ABB RobotStudio station: Practica2_ej2_extra1.rspag

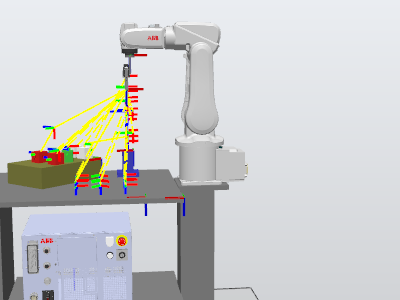
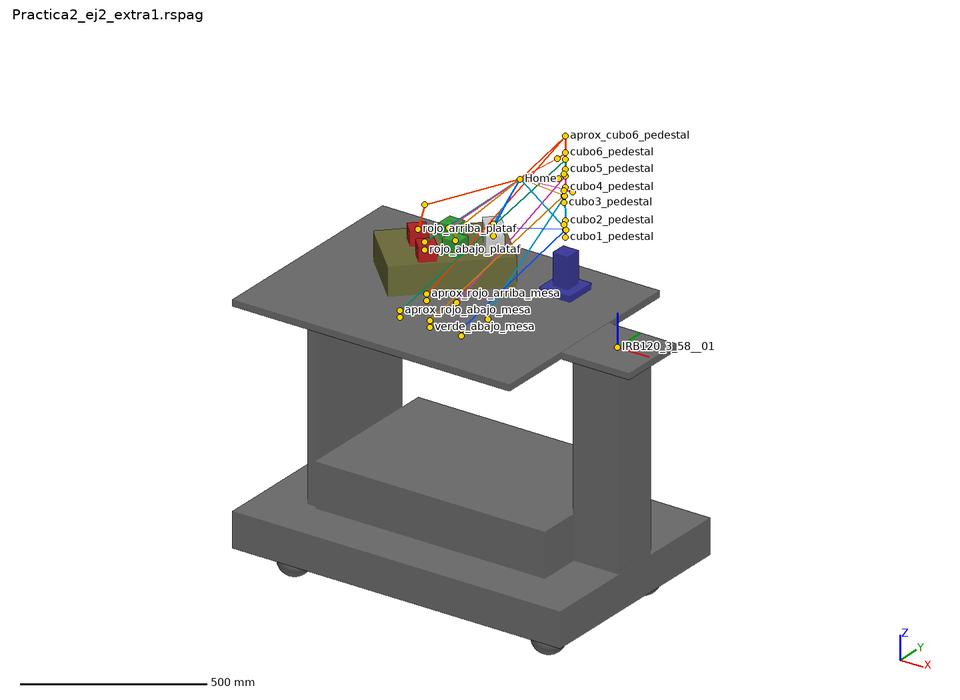
[picture v1: parts stored in the station drawn from their meshes, with robot base, taught points and paths (robot models come from the ABB library and are not in the file)]
--- station ---
Station Practica2_1920 (saved by RobotStudio 24.4.11080.0)
Controller Controlador_IRC5, task T_ROB1: task frame (RAPID world) sits at (560, 0, 840) mm, rotated rx 0 ry 0 rz 180 deg in the station
Controller Controlador_IRC5
  mechanical unit ROB_1: IRB120_3_58__01, 6 joints, base frame (0, 0, 0) mm
Layout (positions relative to the parent item):
  - Pinza_schunk_SGB50 [mechanism, from Libraries\Pinza_schunk_SGB50.rslib] at (258, 0, 1398) mm, rotated rx 180 ry 0 rz 0 deg; joint values [0, 0.1745, -0.1745] (rad or m)
  - Mesa del robot [part], size 1127.5 x 700 x 840 mm
  - Cubo XYZ 50 mm 2 [part] at (-54.74, 116.46, 930) mm, rotated rx 0 ry 0 rz 90 deg, size 50 x 50 x 50 mm
  - Cubo XYZ 50 mm 3 [part] at (7.57, 171.09, 931.86) mm, rotated rx 0 ry 0 rz 45 deg, size 50 x 50 x 50 mm
  - Cubo XYZ 50 mm 4 [part] at (-100.89, 1.6, 929.03) mm, rotated rx 0 ry 0 rz -45 deg, size 50 x 50 x 50 mm
  - Cubo XYZ 50 mm 5 [part] at (5.14, 45.89, 928.53) mm, rotated rx 0 ry 0 rz 90 deg, size 50 x 50 x 50 mm
  - Cubo XYZ 50 mm 6 [part] at (54.86, 109.05, 933.24) mm, rotated rx 0 ry 0 rz 45 deg, size 50 x 50 x 50 mm
  - Cubo XYZ 50 mm 1 [part] at (-175.7, 68.89, 928.24) mm, rotated rx 0 ry 0 rz -45 deg, size 50 x 50 x 50 mm
  - Soporte para elevar los cubos  [part] at (200, 150, 840) mm, size 100 x 100 x 120 mm
  - IRC5_Compact [part, from %ABB.RobotStudio.Models.IRC5%\IRC5_Compact__02.rslib] at (-200, -200, 350) mm
  - Soporte para el controlador [part], size 750 x 480 x 150 mm
  - IRB120_3_58__01 [mechanism, from %ABB.RobotStudio.Models.IRB120%\IRB120_3_58_G_01.rslib] at (560, 0, 840) mm, rotated rx 0 ry 0 rz 180 deg; joint values [0, 0, 0, 0, 1.5708, 0] (rad or m)
  - caja [part], size 406.6 x 406.6 x 90 mm
Attachment: Soporte para el controlador is attached to Mesa del robot
Attachment: Pinza_schunk_SGB50 is attached to IRB120_3_58__01 / Link6
EventTableEntry 2988: Group=, Trigger=D16_O 2989, Actions=[EventTableActionMechanicalPose 2990, EventTableActionAttach 2991], Comment=, ActivationMode=2, Cyclic=false
EventTableTriggerIO 2989: IOValue=[1], IRC5Controller=? -1, Operator=0, SignalSource=Controlador_IRC5 2505
EventTableActionMechanicalPose 2990: VirtualSignal=, Mechanism=Pinza_schunk_SGB50 1474, ToPoseName=HomePosition, VirtualSignalValue=[1]
EventTableActionAttach 2991: AttachmentParent=Pinza_schunk_SGB50 1474, AttachmentChild=? -1, MountObject=false, Offset=[X=1, Y=0, Z=0, W=0, X=0, Y=1, Z=0, W=0, X=0, Y=0, Z=1, W=0, X=0, Y=0, Z=0, W=1], FlangeIndext=0, FindNearest=true
EventTableEntry 2992: Group=, Trigger=D16_O 2993, Actions=[EventTableActionMechanicalPose 2994, EventTableActionDetach 2995], Comment=, ActivationMode=2, Cyclic=false
EventTableTriggerIO 2993: IOValue=[0], IRC5Controller=? -1, Operator=0, SignalSource=Controlador_IRC5 2505
EventTableActionMechanicalPose 2994: VirtualSignal=, Mechanism=Pinza_schunk_SGB50 1474, ToPoseName=Abierto, VirtualSignalValue=[1]
EventTableActionDetach 2995: AttachmentParent=Pinza_schunk_SGB50 1474, AttachmentChild=? -1
EventTableTriggerIO 3053: IOValue=[1], IRC5Controller=? -1, Operator=0, SignalSource=Controlador_IRC5 2505
EventTableTriggerIO 3054: IOValue=[1], IRC5Controller=? -1, Operator=0, SignalSource=Controlador_IRC5 2505
EventTableTriggerIO 3055: IOValue=[1], IRC5Controller=? -1, Operator=0, SignalSource=Controlador_IRC5 2505
EventTableTriggerIO 3056: IOValue=[1], IRC5Controller=? -1, Operator=0, SignalSource=Controlador_IRC5 2505
EventTableTriggerIO 3057: IOValue=[1], IRC5Controller=? -1, Operator=0, SignalSource=Controlador_IRC5 2505
EventTableTriggerIO 3058: IOValue=[1], IRC5Controller=? -1, Operator=0, SignalSource=Controlador_IRC5 2505
EventTableTriggerIO 3059: IOValue=[1], IRC5Controller=? -1, Operator=0, SignalSource=Controlador_IRC5 2505
EventTableTriggerIO 3060: IOValue=[1], IRC5Controller=? -1, Operator=0, SignalSource=Controlador_IRC5 2505
EventTableTriggerIO 3061: IOValue=[1], IRC5Controller=? -1, Operator=0, SignalSource=Controlador_IRC5 2505
EventTableTriggerIO 3062: IOValue=[1], IRC5Controller=? -1, Operator=0, SignalSource=Controlador_IRC5 2505
EventTableTriggerIO 3063: IOValue=[1], IRC5Controller=? -1, Operator=0, SignalSource=Controlador_IRC5 2505
EventTableTriggerIO 3064: IOValue=[1], IRC5Controller=? -1, Operator=0, SignalSource=Controlador_IRC5 2505
EventTableTriggerIO 3065: IOValue=[0], IRC5Controller=? -1, Operator=0, SignalSource=Controlador_IRC5 2505
EventTableTriggerIO 3066: IOValue=[0], IRC5Controller=? -1, Operator=0, SignalSource=Controlador_IRC5 2505
EventTableTriggerIO 3067: IOValue=[0], IRC5Controller=? -1, Operator=0, SignalSource=Controlador_IRC5 2505
EventTableTriggerIO 3068: IOValue=[0], IRC5Controller=? -1, Operator=0, SignalSource=Controlador_IRC5 2505
EventTableTriggerIO 3069: IOValue=[0], IRC5Controller=? -1, Operator=0, SignalSource=Controlador_IRC5 2505
EventTableTriggerIO 3070: IOValue=[0], IRC5Controller=? -1, Operator=0, SignalSource=Controlador_IRC5 2505
EventTableTriggerIO 3071: IOValue=[0], IRC5Controller=? -1, Operator=0, SignalSource=Controlador_IRC5 2505
EventTableTriggerIO 3072: IOValue=[0], IRC5Controller=? -1, Operator=0, SignalSource=Controlador_IRC5 2505
EventTableTriggerIO 3073: IOValue=[0], IRC5Controller=? -1, Operator=0, SignalSource=Controlador_IRC5 2505
EventTableTriggerIO 3074: IOValue=[0], IRC5Controller=? -1, Operator=0, SignalSource=Controlador_IRC5 2505
EventTableTriggerIO 3075: IOValue=[0], IRC5Controller=? -1, Operator=0, SignalSource=Controlador_IRC5 2505
EventTableTriggerIO 3076: IOValue=[0], IRC5Controller=? -1, Operator=0, SignalSource=Controlador_IRC5 2505
EventTableTriggerIO 3176: IOValue=[1], IRC5Controller=? -1, Operator=0, SignalSource=Controlador_IRC5 2505
EventTableTriggerIO 3177: IOValue=[1], IRC5Controller=? -1, Operator=0, SignalSource=Controlador_IRC5 2505
EventTableTriggerIO 3178: IOValue=[1], IRC5Controller=? -1, Operator=0, SignalSource=Controlador_IRC5 2505
EventTableTriggerIO 3179: IOValue=[1], IRC5Controller=? -1, Operator=0, SignalSource=Controlador_IRC5 2505
EventTableTriggerIO 3180: IOValue=[1], IRC5Controller=? -1, Operator=0, SignalSource=Controlador_IRC5 2505
EventTableTriggerIO 3181: IOValue=[0], IRC5Controller=? -1, Operator=0, SignalSource=Controlador_IRC5 2505
EventTableTriggerIO 3182: IOValue=[0], IRC5Controller=? -1, Operator=0, SignalSource=Controlador_IRC5 2505
EventTableTriggerIO 3183: IOValue=[0], IRC5Controller=? -1, Operator=0, SignalSource=Controlador_IRC5 2505
EventTableTriggerIO 3184: IOValue=[0], IRC5Controller=? -1, Operator=0, SignalSource=Controlador_IRC5 2505
EventTableTriggerIO 3185: IOValue=[0], IRC5Controller=? -1, Operator=0, SignalSource=Controlador_IRC5 2505
EventTableTriggerIO 3333: IOValue=[1], IRC5Controller=? -1, Operator=0, SignalSource=Controlador_IRC5 2505
EventTableTriggerIO 3334: IOValue=[1], IRC5Controller=? -1, Operator=0, SignalSource=Controlador_IRC5 2505
EventTableTriggerIO 3335: IOValue=[1], IRC5Controller=? -1, Operator=0, SignalSource=Controlador_IRC5 2505
EventTableTriggerIO 3336: IOValue=[1], IRC5Controller=? -1, Operator=0, SignalSource=Controlador_IRC5 2505
EventTableTriggerIO 3337: IOValue=[1], IRC5Controller=? -1, Operator=0, SignalSource=Controlador_IRC5 2505
EventTableTriggerIO 3338: IOValue=[1], IRC5Controller=? -1, Operator=0, SignalSource=Controlador_IRC5 2505
EventTableTriggerIO 3339: IOValue=[0], IRC5Controller=? -1, Operator=0, SignalSource=Controlador_IRC5 2505
EventTableTriggerIO 3340: IOValue=[0], IRC5Controller=? -1, Operator=0, SignalSource=Controlador_IRC5 2505
EventTableTriggerIO 3341: IOValue=[0], IRC5Controller=? -1, Operator=0, SignalSource=Controlador_IRC5 2505
EventTableTriggerIO 3342: IOValue=[0], IRC5Controller=? -1, Operator=0, SignalSource=Controlador_IRC5 2505
EventTableTriggerIO 3343: IOValue=[0], IRC5Controller=? -1, Operator=0, SignalSource=Controlador_IRC5 2505
EventTableTriggerIO 3344: IOValue=[0], IRC5Controller=? -1, Operator=0, SignalSource=Controlador_IRC5 2505
EventTableTriggerIO 3580: IOValue=[1], IRC5Controller=? -1, Operator=0, SignalSource=Controlador_IRC5 2505
EventTableTriggerIO 3581: IOValue=[1], IRC5Controller=? -1, Operator=0, SignalSource=Controlador_IRC5 2505
EventTableTriggerIO 3582: IOValue=[1], IRC5Controller=? -1, Operator=0, SignalSource=Controlador_IRC5 2505
EventTableTriggerIO 3583: IOValue=[1], IRC5Controller=? -1, Operator=0, SignalSource=Controlador_IRC5 2505
EventTableTriggerIO 3584: IOValue=[1], IRC5Controller=? -1, Operator=0, SignalSource=Controlador_IRC5 2505
EventTableTriggerIO 3585: IOValue=[1], IRC5Controller=? -1, Operator=0, SignalSource=Controlador_IRC5 2505
EventTableTriggerIO 3586: IOValue=[1], IRC5Controller=? -1, Operator=0, SignalSource=Controlador_IRC5 2505
EventTableTriggerIO 3587: IOValue=[1], IRC5Controller=? -1, Operator=0, SignalSource=Controlador_IRC5 2505
EventTableTriggerIO 3588: IOValue=[1], IRC5Controller=? -1, Operator=0, SignalSource=Controlador_IRC5 2505
EventTableTriggerIO 3589: IOValue=[1], IRC5Controller=? -1, Operator=0, SignalSource=Controlador_IRC5 2505
EventTableTriggerIO 3590: IOValue=[0], IRC5Controller=? -1, Operator=0, SignalSource=Controlador_IRC5 2505
EventTableTriggerIO 3591: IOValue=[0], IRC5Controller=? -1, Operator=0, SignalSource=Controlador_IRC5 2505
EventTableTriggerIO 3592: IOValue=[0], IRC5Controller=? -1, Operator=0, SignalSource=Controlador_IRC5 2505
EventTableTriggerIO 3593: IOValue=[0], IRC5Controller=? -1, Operator=0, SignalSource=Controlador_IRC5 2505
EventTableTriggerIO 3594: IOValue=[0], IRC5Controller=? -1, Operator=0, SignalSource=Controlador_IRC5 2505
EventTableTriggerIO 3595: IOValue=[0], IRC5Controller=? -1, Operator=0, SignalSource=Controlador_IRC5 2505
EventTableTriggerIO 3596: IOValue=[0], IRC5Controller=? -1, Operator=0, SignalSource=Controlador_IRC5 2505
EventTableTriggerIO 3597: IOValue=[0], IRC5Controller=? -1, Operator=0, SignalSource=Controlador_IRC5 2505
EventTableTriggerIO 3598: IOValue=[0], IRC5Controller=? -1, Operator=0, SignalSource=Controlador_IRC5 2505
EventTableTriggerIO 3599: IOValue=[0], IRC5Controller=? -1, Operator=0, SignalSource=Controlador_IRC5 2505
EventTableTriggerIO 3839: IOValue=[1], IRC5Controller=? -1, Operator=0, SignalSource=Controlador_IRC5 2505
EventTableTriggerIO 3840: IOValue=[1], IRC5Controller=? -1, Operator=0, SignalSource=Controlador_IRC5 2505
EventTableTriggerIO 3841: IOValue=[1], IRC5Controller=? -1, Operator=0, SignalSource=Controlador_IRC5 2505
EventTableTriggerIO 3842: IOValue=[1], IRC5Controller=? -1, Operator=0, SignalSource=Controlador_IRC5 2505
EventTableTriggerIO 3843: IOValue=[1], IRC5Controller=? -1, Operator=0, SignalSource=Controlador_IRC5 2505
EventTableTriggerIO 3844: IOValue=[1], IRC5Controller=? -1, Operator=0, SignalSource=Controlador_IRC5 2505
EventTableTriggerIO 3845: IOValue=[1], IRC5Controller=? -1, Operator=0, SignalSource=Controlador_IRC5 2505
EventTableTriggerIO 3846: IOValue=[1], IRC5Controller=? -1, Operator=0, SignalSource=Controlador_IRC5 2505
EventTableTriggerIO 3847: IOValue=[1], IRC5Controller=? -1, Operator=0, SignalSource=Controlador_IRC5 2505
EventTableTriggerIO 3848: IOValue=[1], IRC5Controller=? -1, Operator=0, SignalSource=Controlador_IRC5 2505
EventTableTriggerIO 3849: IOValue=[1], IRC5Controller=? -1, Operator=0, SignalSource=Controlador_IRC5 2505
EventTableTriggerIO 3850: IOValue=[1], IRC5Controller=? -1, Operator=0, SignalSource=Controlador_IRC5 2505
EventTableTriggerIO 3851: IOValue=[1], IRC5Controller=? -1, Operator=0, SignalSource=Controlador_IRC5 2505
EventTableTriggerIO 3852: IOValue=[1], IRC5Controller=? -1, Operator=0, SignalSource=Controlador_IRC5 2505
EventTableTriggerIO 3853: IOValue=[1], IRC5Controller=? -1, Operator=0, SignalSource=Controlador_IRC5 2505
EventTableTriggerIO 3854: IOValue=[0], IRC5Controller=? -1, Operator=0, SignalSource=Controlador_IRC5 2505
EventTableTriggerIO 3855: IOValue=[0], IRC5Controller=? -1, Operator=0, SignalSource=Controlador_IRC5 2505
EventTableTriggerIO 3856: IOValue=[0], IRC5Controller=? -1, Operator=0, SignalSource=Controlador_IRC5 2505
EventTableTriggerIO 3857: IOValue=[0], IRC5Controller=? -1, Operator=0, SignalSource=Controlador_IRC5 2505
EventTableTriggerIO 3858: IOValue=[0], IRC5Controller=? -1, Operator=0, SignalSource=Controlador_IRC5 2505
EventTableTriggerIO 3859: IOValue=[0], IRC5Controller=? -1, Operator=0, SignalSource=Controlador_IRC5 2505
EventTableTriggerIO 3860: IOValue=[0], IRC5Controller=? -1, Operator=0, SignalSource=Controlador_IRC5 2505
EventTableTriggerIO 3861: IOValue=[0], IRC5Controller=? -1, Operator=0, SignalSource=Controlador_IRC5 2505
EventTableTriggerIO 3862: IOValue=[0], IRC5Controller=? -1, Operator=0, SignalSource=Controlador_IRC5 2505
EventTableTriggerIO 3863: IOValue=[0], IRC5Controller=? -1, Operator=0, SignalSource=Controlador_IRC5 2505
EventTableTriggerIO 3864: IOValue=[0], IRC5Controller=? -1, Operator=0, SignalSource=Controlador_IRC5 2505
EventTableTriggerIO 3865: IOValue=[0], IRC5Controller=? -1, Operator=0, SignalSource=Controlador_IRC5 2505
EventTableTriggerIO 3866: IOValue=[0], IRC5Controller=? -1, Operator=0, SignalSource=Controlador_IRC5 2505
EventTableTriggerIO 3867: IOValue=[0], IRC5Controller=? -1, Operator=0, SignalSource=Controlador_IRC5 2505
EventTableTriggerIO 3868: IOValue=[0], IRC5Controller=? -1, Operator=0, SignalSource=Controlador_IRC5 2505
EventTableTriggerIO 4020: IOValue=[1], IRC5Controller=? -1, Operator=0, SignalSource=Controlador_IRC5 2505
EventTableTriggerIO 4021: IOValue=[1], IRC5Controller=? -1, Operator=0, SignalSource=Controlador_IRC5 2505
EventTableTriggerIO 4022: IOValue=[1], IRC5Controller=? -1, Operator=0, SignalSource=Controlador_IRC5 2505
EventTableTriggerIO 4023: IOValue=[1], IRC5Controller=? -1, Operator=0, SignalSource=Controlador_IRC5 2505
EventTableTriggerIO 4024: IOValue=[1], IRC5Controller=? -1, Operator=0, SignalSource=Controlador_IRC5 2505
EventTableTriggerIO 4025: IOValue=[1], IRC5Controller=? -1, Operator=0, SignalSource=Controlador_IRC5 2505
EventTableTriggerIO 4026: IOValue=[0], IRC5Controller=? -1, Operator=0, SignalSource=Controlador_IRC5 2505
EventTableTriggerIO 4027: IOValue=[0], IRC5Controller=? -1, Operator=0, SignalSource=Controlador_IRC5 2505
EventTableTriggerIO 4028: IOValue=[0], IRC5Controller=? -1, Operator=0, SignalSource=Controlador_IRC5 2505
EventTableTriggerIO 4029: IOValue=[0], IRC5Controller=? -1, Operator=0, SignalSource=Controlador_IRC5 2505
EventTableTriggerIO 4030: IOValue=[0], IRC5Controller=? -1, Operator=0, SignalSource=Controlador_IRC5 2505
EventTableTriggerIO 4031: IOValue=[0], IRC5Controller=? -1, Operator=0, SignalSource=Controlador_IRC5 2505
EventTableTriggerIO 4133: IOValue=[1], IRC5Controller=? -1, Operator=0, SignalSource=Controlador_IRC5 2505
EventTableTriggerIO 4134: IOValue=[1], IRC5Controller=? -1, Operator=0, SignalSource=Controlador_IRC5 2505
EventTableTriggerIO 4135: IOValue=[0], IRC5Controller=? -1, Operator=0, SignalSource=Controlador_IRC5 2505
EventTableTriggerIO 4136: IOValue=[0], IRC5Controller=? -1, Operator=0, SignalSource=Controlador_IRC5 2505
EventTableTriggerIO 4229: IOValue=[1], IRC5Controller=? -1, Operator=0, SignalSource=Controlador_IRC5 2505
EventTableTriggerIO 4230: IOValue=[1], IRC5Controller=? -1, Operator=0, SignalSource=Controlador_IRC5 2505
EventTableTriggerIO 4231: IOValue=[1], IRC5Controller=? -1, Operator=0, SignalSource=Controlador_IRC5 2505
EventTableTriggerIO 4232: IOValue=[1], IRC5Controller=? -1, Operator=0, SignalSource=Controlador_IRC5 2505
EventTableTriggerIO 4233: IOValue=[1], IRC5Controller=? -1, Operator=0, SignalSource=Controlador_IRC5 2505
EventTableTriggerIO 4234: IOValue=[1], IRC5Controller=? -1, Operator=0, SignalSource=Controlador_IRC5 2505
EventTableTriggerIO 4235: IOValue=[0], IRC5Controller=? -1, Operator=0, SignalSource=Controlador_IRC5 2505
EventTableTriggerIO 4236: IOValue=[0], IRC5Controller=? -1, Operator=0, SignalSource=Controlador_IRC5 2505
EventTableTriggerIO 4237: IOValue=[0], IRC5Controller=? -1, Operator=0, SignalSource=Controlador_IRC5 2505
EventTableTriggerIO 4238: IOValue=[0], IRC5Controller=? -1, Operator=0, SignalSource=Controlador_IRC5 2505
EventTableTriggerIO 4239: IOValue=[0], IRC5Controller=? -1, Operator=0, SignalSource=Controlador_IRC5 2505
EventTableTriggerIO 4240: IOValue=[0], IRC5Controller=? -1, Operator=0, SignalSource=Controlador_IRC5 2505
EventTableTriggerIO 4476: IOValue=[1], IRC5Controller=? -1, Operator=0, SignalSource=Controlador_IRC5 2505
EventTableTriggerIO 4477: IOValue=[1], IRC5Controller=? -1, Operator=0, SignalSource=Controlador_IRC5 2505
EventTableTriggerIO 4478: IOValue=[1], IRC5Controller=? -1, Operator=0, SignalSource=Controlador_IRC5 2505
EventTableTriggerIO 4479: IOValue=[1], IRC5Controller=? -1, Operator=0, SignalSource=Controlador_IRC5 2505
EventTableTriggerIO 4480: IOValue=[1], IRC5Controller=? -1, Operator=0, SignalSource=Controlador_IRC5 2505
EventTableTriggerIO 4481: IOValue=[0], IRC5Controller=? -1, Operator=0, SignalSource=Controlador_IRC5 2505
EventTableTriggerIO 4482: IOValue=[0], IRC5Controller=? -1, Operator=0, SignalSource=Controlador_IRC5 2505
EventTableTriggerIO 4483: IOValue=[0], IRC5Controller=? -1, Operator=0, SignalSource=Controlador_IRC5 2505
EventTableTriggerIO 4484: IOValue=[0], IRC5Controller=? -1, Operator=0, SignalSource=Controlador_IRC5 2505
EventTableTriggerIO 4485: IOValue=[0], IRC5Controller=? -1, Operator=0, SignalSource=Controlador_IRC5 2505
EventTableTriggerIO 4657: IOValue=[1], IRC5Controller=? -1, Operator=0, SignalSource=Controlador_IRC5 2505
EventTableTriggerIO 4658: IOValue=[1], IRC5Controller=? -1, Operator=0, SignalSource=Controlador_IRC5 2505
EventTableTriggerIO 4659: IOValue=[1], IRC5Controller=? -1, Operator=0, SignalSource=Controlador_IRC5 2505
EventTableTriggerIO 4660: IOValue=[1], IRC5Controller=? -1, Operator=0, SignalSource=Controlador_IRC5 2505
EventTableTriggerIO 4661: IOValue=[1], IRC5Controller=? -1, Operator=0, SignalSource=Controlador_IRC5 2505
EventTableTriggerIO 4662: IOValue=[0], IRC5Controller=? -1, Operator=0, SignalSource=Controlador_IRC5 2505
EventTableTriggerIO 4663: IOValue=[0], IRC5Controller=? -1, Operator=0, SignalSource=Controlador_IRC5 2505
EventTableTriggerIO 4664: IOValue=[0], IRC5Controller=? -1, Operator=0, SignalSource=Controlador_IRC5 2505
EventTableTriggerIO 4665: IOValue=[0], IRC5Controller=? -1, Operator=0, SignalSource=Controlador_IRC5 2505
EventTableTriggerIO 4666: IOValue=[0], IRC5Controller=? -1, Operator=0, SignalSource=Controlador_IRC5 2505
EventTableTriggerIO 4783: IOValue=[1], IRC5Controller=? -1, Operator=0, SignalSource=Controlador_IRC5 2505
EventTableTriggerIO 4784: IOValue=[1], IRC5Controller=? -1, Operator=0, SignalSource=Controlador_IRC5 2505
EventTableTriggerIO 4785: IOValue=[1], IRC5Controller=? -1, Operator=0, SignalSource=Controlador_IRC5 2505
EventTableTriggerIO 4786: IOValue=[1], IRC5Controller=? -1, Operator=0, SignalSource=Controlador_IRC5 2505
EventTableTriggerIO 4787: IOValue=[1], IRC5Controller=? -1, Operator=0, SignalSource=Controlador_IRC5 2505
EventTableTriggerIO 4788: IOValue=[1], IRC5Controller=? -1, Operator=0, SignalSource=Controlador_IRC5 2505
EventTableTriggerIO 4789: IOValue=[1], IRC5Controller=? -1, Operator=0, SignalSource=Controlador_IRC5 2505
EventTableTriggerIO 4790: IOValue=[1], IRC5Controller=? -1, Operator=0, SignalSource=Controlador_IRC5 2505
EventTableTriggerIO 4791: IOValue=[1], IRC5Controller=? -1, Operator=0, SignalSource=Controlador_IRC5 2505
EventTableTriggerIO 4792: IOValue=[1], IRC5Controller=? -1, Operator=0, SignalSource=Controlador_IRC5 2505
EventTableTriggerIO 4793: IOValue=[1], IRC5Controller=? -1, Operator=0, SignalSource=Controlador_IRC5 2505
EventTableTriggerIO 4794: IOValue=[1], IRC5Controller=? -1, Operator=0, SignalSource=Controlador_IRC5 2505
EventTableTriggerIO 4795: IOValue=[0], IRC5Controller=? -1, Operator=0, SignalSource=Controlador_IRC5 2505
EventTableTriggerIO 4796: IOValue=[0], IRC5Controller=? -1, Operator=0, SignalSource=Controlador_IRC5 2505
EventTableTriggerIO 4797: IOValue=[0], IRC5Controller=? -1, Operator=0, SignalSource=Controlador_IRC5 2505
EventTableTriggerIO 4798: IOValue=[0], IRC5Controller=? -1, Operator=0, SignalSource=Controlador_IRC5 2505
EventTableTriggerIO 4799: IOValue=[0], IRC5Controller=? -1, Operator=0, SignalSource=Controlador_IRC5 2505
EventTableTriggerIO 4800: IOValue=[0], IRC5Controller=? -1, Operator=0, SignalSource=Controlador_IRC5 2505
EventTableTriggerIO 4801: IOValue=[0], IRC5Controller=? -1, Operator=0, SignalSource=Controlador_IRC5 2505
EventTableTriggerIO 4802: IOValue=[0], IRC5Controller=? -1, Operator=0, SignalSource=Controlador_IRC5 2505
EventTableTriggerIO 4803: IOValue=[0], IRC5Controller=? -1, Operator=0, SignalSource=Controlador_IRC5 2505
EventTableTriggerIO 4804: IOValue=[0], IRC5Controller=? -1, Operator=0, SignalSource=Controlador_IRC5 2505
EventTableTriggerIO 4805: IOValue=[0], IRC5Controller=? -1, Operator=0, SignalSource=Controlador_IRC5 2505
EventTableTriggerIO 4806: IOValue=[0], IRC5Controller=? -1, Operator=0, SignalSource=Controlador_IRC5 2505
EventTableTriggerIO 5023: IOValue=[1], IRC5Controller=? -1, Operator=0, SignalSource=Controlador_IRC5 2505
EventTableTriggerIO 5024: IOValue=[1], IRC5Controller=? -1, Operator=0, SignalSource=Controlador_IRC5 2505
EventTableTriggerIO 5025: IOValue=[1], IRC5Controller=? -1, Operator=0, SignalSource=Controlador_IRC5 2505
EventTableTriggerIO 5026: IOValue=[1], IRC5Controller=? -1, Operator=0, SignalSource=Controlador_IRC5 2505
EventTableTriggerIO 5027: IOValue=[1], IRC5Controller=? -1, Operator=0, SignalSource=Controlador_IRC5 2505
EventTableTriggerIO 5028: IOValue=[1], IRC5Controller=? -1, Operator=0, SignalSource=Controlador_IRC5 2505
EventTableTriggerIO 5029: IOValue=[0], IRC5Controller=? -1, Operator=0, SignalSource=Controlador_IRC5 2505
EventTableTriggerIO 5030: IOValue=[0], IRC5Controller=? -1, Operator=0, SignalSource=Controlador_IRC5 2505
EventTableTriggerIO 5031: IOValue=[0], IRC5Controller=? -1, Operator=0, SignalSource=Controlador_IRC5 2505
EventTableTriggerIO 5032: IOValue=[0], IRC5Controller=? -1, Operator=0, SignalSource=Controlador_IRC5 2505
EventTableTriggerIO 5033: IOValue=[0], IRC5Controller=? -1, Operator=0, SignalSource=Controlador_IRC5 2505
EventTableTriggerIO 5034: IOValue=[0], IRC5Controller=? -1, Operator=0, SignalSource=Controlador_IRC5 2505
EventTableTriggerIO 5081: IOValue=[1], IRC5Controller=? -1, Operator=0, SignalSource=Controlador_IRC5 2505
EventTableTriggerIO 5082: IOValue=[1], IRC5Controller=? -1, Operator=0, SignalSource=Controlador_IRC5 2505
EventTableTriggerIO 5083: IOValue=[1], IRC5Controller=? -1, Operator=0, SignalSource=Controlador_IRC5 2505
EventTableTriggerIO 5084: IOValue=[1], IRC5Controller=? -1, Operator=0, SignalSource=Controlador_IRC5 2505
EventTableTriggerIO 5085: IOValue=[1], IRC5Controller=? -1, Operator=0, SignalSource=Controlador_IRC5 2505
EventTableTriggerIO 5086: IOValue=[1], IRC5Controller=? -1, Operator=0, SignalSource=Controlador_IRC5 2505
EventTableTriggerIO 5087: IOValue=[1], IRC5Controller=? -1, Operator=0, SignalSource=Controlador_IRC5 2505
EventTableTriggerIO 5088: IOValue=[0], IRC5Controller=? -1, Operator=0, SignalSource=Controlador_IRC5 2505
EventTableTriggerIO 5089: IOValue=[0], IRC5Controller=? -1, Operator=0, SignalSource=Controlador_IRC5 2505
EventTableTriggerIO 5090: IOValue=[0], IRC5Controller=? -1, Operator=0, SignalSource=Controlador_IRC5 2505
EventTableTriggerIO 5091: IOValue=[0], IRC5Controller=? -1, Operator=0, SignalSource=Controlador_IRC5 2505
EventTableTriggerIO 5092: IOValue=[0], IRC5Controller=? -1, Operator=0, SignalSource=Controlador_IRC5 2505
EventTableTriggerIO 5093: IOValue=[0], IRC5Controller=? -1, Operator=0, SignalSource=Controlador_IRC5 2505
EventTableTriggerIO 5094: IOValue=[0], IRC5Controller=? -1, Operator=0, SignalSource=Controlador_IRC5 2505
EventTableTriggerIO 5236: IOValue=[1], IRC5Controller=? -1, Operator=0, SignalSource=Controlador_IRC5 2505
EventTableTriggerIO 5237: IOValue=[1], IRC5Controller=? -1, Operator=0, SignalSource=Controlador_IRC5 2505
EventTableTriggerIO 5238: IOValue=[1], IRC5Controller=? -1, Operator=0, SignalSource=Controlador_IRC5 2505
EventTableTriggerIO 5239: IOValue=[1], IRC5Controller=? -1, Operator=0, SignalSource=Controlador_IRC5 2505
EventTableTriggerIO 5240: IOValue=[0], IRC5Controller=? -1, Operator=0, SignalSource=Controlador_IRC5 2505
EventTableTriggerIO 5241: IOValue=[0], IRC5Controller=? -1, Operator=0, SignalSource=Controlador_IRC5 2505
EventTableTriggerIO 5242: IOValue=[0], IRC5Controller=? -1, Operator=0, SignalSource=Controlador_IRC5 2505
EventTableTriggerIO 5243: IOValue=[0], IRC5Controller=? -1, Operator=0, SignalSource=Controlador_IRC5 2505
EventTableTriggerIO 5512: IOValue=[1], IRC5Controller=? -1, Operator=0, SignalSource=Controlador_IRC5 2505
EventTableTriggerIO 5513: IOValue=[1], IRC5Controller=? -1, Operator=0, SignalSource=Controlador_IRC5 2505
EventTableTriggerIO 5514: IOValue=[1], IRC5Controller=? -1, Operator=0, SignalSource=Controlador_IRC5 2505
EventTableTriggerIO 5515: IOValue=[1], IRC5Controller=? -1, Operator=0, SignalSource=Controlador_IRC5 2505
EventTableTriggerIO 5516: IOValue=[1], IRC5Controller=? -1, Operator=0, SignalSource=Controlador_IRC5 2505
EventTableTriggerIO 5517: IOValue=[1], IRC5Controller=? -1, Operator=0, SignalSource=Controlador_IRC5 2505
EventTableTriggerIO 5518: IOValue=[1], IRC5Controller=? -1, Operator=0, SignalSource=Controlador_IRC5 2505
EventTableTriggerIO 5519: IOValue=[1], IRC5Controller=? -1, Operator=0, SignalSource=Controlador_IRC5 2505
EventTableTriggerIO 5520: IOValue=[1], IRC5Controller=? -1, Operator=0, SignalSource=Controlador_IRC5 2505
EventTableTriggerIO 5521: IOValue=[1], IRC5Controller=? -1, Operator=0, SignalSource=Controlador_IRC5 2505
EventTableTriggerIO 5522: IOValue=[1], IRC5Controller=? -1, Operator=0, SignalSource=Controlador_IRC5 2505
EventTableTriggerIO 5523: IOValue=[1], IRC5Controller=? -1, Operator=0, SignalSource=Controlador_IRC5 2505
EventTableTriggerIO 5524: IOValue=[1], IRC5Controller=? -1, Operator=0, SignalSource=Controlador_IRC5 2505
EventTableTriggerIO 5525: IOValue=[1], IRC5Controller=? -1, Operator=0, SignalSource=Controlador_IRC5 2505
EventTableTriggerIO 5526: IOValue=[0], IRC5Controller=? -1, Operator=0, SignalSource=Controlador_IRC5 2505
EventTableTriggerIO 5527: IOValue=[0], IRC5Controller=? -1, Operator=0, SignalSource=Controlador_IRC5 2505
EventTableTriggerIO 5528: IOValue=[0], IRC5Controller=? -1, Operator=0, SignalSource=Controlador_IRC5 2505
EventTableTriggerIO 5529: IOValue=[0], IRC5Controller=? -1, Operator=0, SignalSource=Controlador_IRC5 2505
EventTableTriggerIO 5530: IOValue=[0], IRC5Controller=? -1, Operator=0, SignalSource=Controlador_IRC5 2505
EventTableTriggerIO 5531: IOValue=[0], IRC5Controller=? -1, Operator=0, SignalSource=Controlador_IRC5 2505
EventTableTriggerIO 5532: IOValue=[0], IRC5Controller=? -1, Operator=0, SignalSource=Controlador_IRC5 2505
EventTableTriggerIO 5533: IOValue=[0], IRC5Controller=? -1, Operator=0, SignalSource=Controlador_IRC5 2505
EventTableTriggerIO 5534: IOValue=[0], IRC5Controller=? -1, Operator=0, SignalSource=Controlador_IRC5 2505
EventTableTriggerIO 5535: IOValue=[0], IRC5Controller=? -1, Operator=0, SignalSource=Controlador_IRC5 2505
EventTableTriggerIO 5536: IOValue=[0], IRC5Controller=? -1, Operator=0, SignalSource=Controlador_IRC5 2505
EventTableTriggerIO 5537: IOValue=[0], IRC5Controller=? -1, Operator=0, SignalSource=Controlador_IRC5 2505
EventTableTriggerIO 5538: IOValue=[0], IRC5Controller=? -1, Operator=0, SignalSource=Controlador_IRC5 2505
EventTableTriggerIO 5539: IOValue=[0], IRC5Controller=? -1, Operator=0, SignalSource=Controlador_IRC5 2505
EventTableTriggerIO 5657: IOValue=[1], IRC5Controller=? -1, Operator=0, SignalSource=Controlador_IRC5 2505
EventTableTriggerIO 5658: IOValue=[1], IRC5Controller=? -1, Operator=0, SignalSource=Controlador_IRC5 2505
EventTableTriggerIO 5659: IOValue=[1], IRC5Controller=? -1, Operator=0, SignalSource=Controlador_IRC5 2505
EventTableTriggerIO 5660: IOValue=[1], IRC5Controller=? -1, Operator=0, SignalSource=Controlador_IRC5 2505
EventTableTriggerIO 5661: IOValue=[1], IRC5Controller=? -1, Operator=0, SignalSource=Controlador_IRC5 2505
EventTableTriggerIO 5662: IOValue=[1], IRC5Controller=? -1, Operator=0, SignalSource=Controlador_IRC5 2505
EventTableTriggerIO 5663: IOValue=[1], IRC5Controller=? -1, Operator=0, SignalSource=Controlador_IRC5 2505
EventTableTriggerIO 5664: IOValue=[1], IRC5Controller=? -1, Operator=0, SignalSource=Controlador_IRC5 2505
EventTableTriggerIO 5665: IOValue=[1], IRC5Controller=? -1, Operator=0, SignalSource=Controlador_IRC5 2505
EventTableTriggerIO 5666: IOValue=[1], IRC5Controller=? -1, Operator=0, SignalSource=Controlador_IRC5 2505
EventTableTriggerIO 5667: IOValue=[1], IRC5Controller=? -1, Operator=0, SignalSource=Controlador_IRC5 2505
EventTableTriggerIO 5668: IOValue=[1], IRC5Controller=? -1, Operator=0, SignalSource=Controlador_IRC5 2505
EventTableTriggerIO 5669: IOValue=[1], IRC5Controller=? -1, Operator=0, SignalSource=Controlador_IRC5 2505
EventTableTriggerIO 5670: IOValue=[1], IRC5Controller=? -1, Operator=0, SignalSource=Controlador_IRC5 2505
EventTableTriggerIO 5671: IOValue=[1], IRC5Controller=? -1, Operator=0, SignalSource=Controlador_IRC5 2505
EventTableTriggerIO 5672: IOValue=[1], IRC5Controller=? -1, Operator=0, SignalSource=Controlador_IRC5 2505
EventTableTriggerIO 5673: IOValue=[1], IRC5Controller=? -1, Operator=0, SignalSource=Controlador_IRC5 2505
EventTableTriggerIO 5674: IOValue=[1], IRC5Controller=? -1, Operator=0, SignalSource=Controlador_IRC5 2505
EventTableTriggerIO 5675: IOValue=[1], IRC5Controller=? -1, Operator=0, SignalSource=Controlador_IRC5 2505
EventTableTriggerIO 5676: IOValue=[1], IRC5Controller=? -1, Operator=0, SignalSource=Controlador_IRC5 2505
EventTableTriggerIO 5677: IOValue=[1], IRC5Controller=? -1, Operator=0, SignalSource=Controlador_IRC5 2505
EventTableTriggerIO 5678: IOValue=[1], IRC5Controller=? -1, Operator=0, SignalSource=Controlador_IRC5 2505
EventTableTriggerIO 5679: IOValue=[0], IRC5Controller=? -1, Operator=0, SignalSource=Controlador_IRC5 2505
EventTableTriggerIO 5680: IOValue=[0], IRC5Controller=? -1, Operator=0, SignalSource=Controlador_IRC5 2505
EventTableTriggerIO 5681: IOValue=[0], IRC5Controller=? -1, Operator=0, SignalSource=Controlador_IRC5 2505
EventTableTriggerIO 5682: IOValue=[0], IRC5Controller=? -1, Operator=0, SignalSource=Controlador_IRC5 2505
EventTableTriggerIO 5683: IOValue=[0], IRC5Controller=? -1, Operator=0, SignalSource=Controlador_IRC5 2505
EventTableTriggerIO 5684: IOValue=[0], IRC5Controller=? -1, Operator=0, SignalSource=Controlador_IRC5 2505
EventTableTriggerIO 5685: IOValue=[0], IRC5Controller=? -1, Operator=0, SignalSource=Controlador_IRC5 2505
EventTableTriggerIO 5686: IOValue=[0], IRC5Controller=? -1, Operator=0, SignalSource=Controlador_IRC5 2505
EventTableTriggerIO 5687: IOValue=[0], IRC5Controller=? -1, Operator=0, SignalSource=Controlador_IRC5 2505
EventTableTriggerIO 5688: IOValue=[0], IRC5Controller=? -1, Operator=0, SignalSource=Controlador_IRC5 2505
EventTableTriggerIO 5689: IOValue=[0], IRC5Controller=? -1, Operator=0, SignalSource=Controlador_IRC5 2505
EventTableTriggerIO 5690: IOValue=[0], IRC5Controller=? -1, Operator=0, SignalSource=Controlador_IRC5 2505
EventTableTriggerIO 5691: IOValue=[0], IRC5Controller=? -1, Operator=0, SignalSource=Controlador_IRC5 2505
EventTableTriggerIO 5692: IOValue=[0], IRC5Controller=? -1, Operator=0, SignalSource=Controlador_IRC5 2505
EventTableTriggerIO 5693: IOValue=[0], IRC5Controller=? -1, Operator=0, SignalSource=Controlador_IRC5 2505
EventTableTriggerIO 5694: IOValue=[0], IRC5Controller=? -1, Operator=0, SignalSource=Controlador_IRC5 2505
EventTableTriggerIO 5695: IOValue=[0], IRC5Controller=? -1, Operator=0, SignalSource=Controlador_IRC5 2505
EventTableTriggerIO 5696: IOValue=[0], IRC5Controller=? -1, Operator=0, SignalSource=Controlador_IRC5 2505
EventTableTriggerIO 5697: IOValue=[0], IRC5Controller=? -1, Operator=0, SignalSource=Controlador_IRC5 2505
EventTableTriggerIO 5698: IOValue=[0], IRC5Controller=? -1, Operator=0, SignalSource=Controlador_IRC5 2505
EventTableTriggerIO 5699: IOValue=[0], IRC5Controller=? -1, Operator=0, SignalSource=Controlador_IRC5 2505
EventTableTriggerIO 5700: IOValue=[0], IRC5Controller=? -1, Operator=0, SignalSource=Controlador_IRC5 2505
EventTableTriggerIO 5755: IOValue=[1], IRC5Controller=? -1, Operator=0, SignalSource=Controlador_IRC5 2505
EventTableTriggerIO 5756: IOValue=[1], IRC5Controller=? -1, Operator=0, SignalSource=Controlador_IRC5 2505
EventTableTriggerIO 5757: IOValue=[1], IRC5Controller=? -1, Operator=0, SignalSource=Controlador_IRC5 2505
EventTableTriggerIO 5758: IOValue=[1], IRC5Controller=? -1, Operator=0, SignalSource=Controlador_IRC5 2505
EventTableTriggerIO 5759: IOValue=[1], IRC5Controller=? -1, Operator=0, SignalSource=Controlador_IRC5 2505
EventTableTriggerIO 5760: IOValue=[1], IRC5Controller=? -1, Operator=0, SignalSource=Controlador_IRC5 2505
EventTableTriggerIO 5761: IOValue=[1], IRC5Controller=? -1, Operator=0, SignalSource=Controlador_IRC5 2505
EventTableTriggerIO 5762: IOValue=[1], IRC5Controller=? -1, Operator=0, SignalSource=Controlador_IRC5 2505
EventTableTriggerIO 5763: IOValue=[1], IRC5Controller=? -1, Operator=0, SignalSource=Controlador_IRC5 2505
EventTableTriggerIO 5764: IOValue=[1], IRC5Controller=? -1, Operator=0, SignalSource=Controlador_IRC5 2505
EventTableTriggerIO 5765: IOValue=[1], IRC5Controller=? -1, Operator=0, SignalSource=Controlador_IRC5 2505
EventTableTriggerIO 5766: IOValue=[0], IRC5Controller=? -1, Operator=0, SignalSource=Controlador_IRC5 2505
EventTableTriggerIO 5767: IOValue=[0], IRC5Controller=? -1, Operator=0, SignalSource=Controlador_IRC5 2505
EventTableTriggerIO 5768: IOValue=[0], IRC5Controller=? -1, Operator=0, SignalSource=Controlador_IRC5 2505
EventTableTriggerIO 5769: IOValue=[0], IRC5Controller=? -1, Operator=0, SignalSource=Controlador_IRC5 2505
EventTableTriggerIO 5770: IOValue=[0], IRC5Controller=? -1, Operator=0, SignalSource=Controlador_IRC5 2505
EventTableTriggerIO 5771: IOValue=[0], IRC5Controller=? -1, Operator=0, SignalSource=Controlador_IRC5 2505
EventTableTriggerIO 5772: IOValue=[0], IRC5Controller=? -1, Operator=0, SignalSource=Controlador_IRC5 2505
EventTableTriggerIO 5773: IOValue=[0], IRC5Controller=? -1, Operator=0, SignalSource=Controlador_IRC5 2505
EventTableTriggerIO 5774: IOValue=[0], IRC5Controller=? -1, Operator=0, SignalSource=Controlador_IRC5 2505
EventTableTriggerIO 5775: IOValue=[0], IRC5Controller=? -1, Operator=0, SignalSource=Controlador_IRC5 2505
EventTableTriggerIO 5776: IOValue=[0], IRC5Controller=? -1, Operator=0, SignalSource=Controlador_IRC5 2505
EventTableTriggerIO 5791: IOValue=[1], IRC5Controller=? -1, Operator=0, SignalSource=Controlador_IRC5 2505
EventTableTriggerIO 5792: IOValue=[1], IRC5Controller=? -1, Operator=0, SignalSource=Controlador_IRC5 2505
EventTableTriggerIO 5793: IOValue=[1], IRC5Controller=? -1, Operator=0, SignalSource=Controlador_IRC5 2505
EventTableTriggerIO 5794: IOValue=[1], IRC5Controller=? -1, Operator=0, SignalSource=Controlador_IRC5 2505
EventTableTriggerIO 5795: IOValue=[1], IRC5Controller=? -1, Operator=0, SignalSource=Controlador_IRC5 2505
EventTableTriggerIO 5796: IOValue=[1], IRC5Controller=? -1, Operator=0, SignalSource=Controlador_IRC5 2505
EventTableTriggerIO 5797: IOValue=[1], IRC5Controller=? -1, Operator=0, SignalSource=Controlador_IRC5 2505
EventTableTriggerIO 5798: IOValue=[1], IRC5Controller=? -1, Operator=0, SignalSource=Controlador_IRC5 2505
EventTableTriggerIO 5799: IOValue=[1], IRC5Controller=? -1, Operator=0, SignalSource=Controlador_IRC5 2505
EventTableTriggerIO 5800: IOValue=[1], IRC5Controller=? -1, Operator=0, SignalSource=Controlador_IRC5 2505
EventTableTriggerIO 5801: IOValue=[1], IRC5Controller=? -1, Operator=0, SignalSource=Controlador_IRC5 2505
EventTableTriggerIO 5802: IOValue=[1], IRC5Controller=? -1, Operator=0, SignalSource=Controlador_IRC5 2505
EventTableTriggerIO 5803: IOValue=[1], IRC5Controller=? -1, Operator=0, SignalSource=Controlador_IRC5 2505
EventTableTriggerIO 5804: IOValue=[0], IRC5Controller=? -1, Operator=0, SignalSource=Controlador_IRC5 2505
EventTableTriggerIO 5805: IOValue=[0], IRC5Controller=? -1, Operator=0, SignalSource=Controlador_IRC5 2505
EventTableTriggerIO 5806: IOValue=[0], IRC5Controller=? -1, Operator=0, SignalSource=Controlador_IRC5 2505
EventTableTriggerIO 5807: IOValue=[0], IRC5Controller=? -1, Operator=0, SignalSource=Controlador_IRC5 2505
EventTableTriggerIO 5808: IOValue=[0], IRC5Controller=? -1, Operator=0, SignalSource=Controlador_IRC5 2505
EventTableTriggerIO 5809: IOValue=[0], IRC5Controller=? -1, Operator=0, SignalSource=Controlador_IRC5 2505
EventTableTriggerIO 5810: IOValue=[0], IRC5Controller=? -1, Operator=0, SignalSource=Controlador_IRC5 2505
EventTableTriggerIO 5811: IOValue=[0], IRC5Controller=? -1, Operator=0, SignalSource=Controlador_IRC5 2505
EventTableTriggerIO 5812: IOValue=[0], IRC5Controller=? -1, Operator=0, SignalSource=Controlador_IRC5 2505
EventTableTriggerIO 5813: IOValue=[0], IRC5Controller=? -1, Operator=0, SignalSource=Controlador_IRC5 2505
EventTableTriggerIO 5814: IOValue=[0], IRC5Controller=? -1, Operator=0, SignalSource=Controlador_IRC5 2505
EventTableTriggerIO 5815: IOValue=[0], IRC5Controller=? -1, Operator=0, SignalSource=Controlador_IRC5 2505
EventTableTriggerIO 5816: IOValue=[0], IRC5Controller=? -1, Operator=0, SignalSource=Controlador_IRC5 2505
EventTableTriggerIO 5842: IOValue=[1], IRC5Controller=? -1, Operator=0, SignalSource=Controlador_IRC5 2505
EventTableTriggerIO 5843: IOValue=[1], IRC5Controller=? -1, Operator=0, SignalSource=Controlador_IRC5 2505
EventTableTriggerIO 5844: IOValue=[1], IRC5Controller=? -1, Operator=0, SignalSource=Controlador_IRC5 2505
EventTableTriggerIO 5845: IOValue=[0], IRC5Controller=? -1, Operator=0, SignalSource=Controlador_IRC5 2505
EventTableTriggerIO 5846: IOValue=[0], IRC5Controller=? -1, Operator=0, SignalSource=Controlador_IRC5 2505
EventTableTriggerIO 5847: IOValue=[0], IRC5Controller=? -1, Operator=0, SignalSource=Controlador_IRC5 2505
EventTableTriggerIO 5854: IOValue=[1], IRC5Controller=? -1, Operator=0, SignalSource=Controlador_IRC5 2505
EventTableTriggerIO 5855: IOValue=[1], IRC5Controller=? -1, Operator=0, SignalSource=Controlador_IRC5 2505
EventTableTriggerIO 5856: IOValue=[1], IRC5Controller=? -1, Operator=0, SignalSource=Controlador_IRC5 2505
EventTableTriggerIO 5857: IOValue=[1], IRC5Controller=? -1, Operator=0, SignalSource=Controlador_IRC5 2505
EventTableTriggerIO 5858: IOValue=[1], IRC5Controller=? -1, Operator=0, SignalSource=Controlador_IRC5 2505
EventTableTriggerIO 5859: IOValue=[0], IRC5Controller=? -1, Operator=0, SignalSource=Controlador_IRC5 2505
EventTableTriggerIO 5860: IOValue=[0], IRC5Controller=? -1, Operator=0, SignalSource=Controlador_IRC5 2505
EventTableTriggerIO 5861: IOValue=[0], IRC5Controller=? -1, Operator=0, SignalSource=Controlador_IRC5 2505
EventTableTriggerIO 5862: IOValue=[0], IRC5Controller=? -1, Operator=0, SignalSource=Controlador_IRC5 2505
EventTableTriggerIO 5863: IOValue=[0], IRC5Controller=? -1, Operator=0, SignalSource=Controlador_IRC5 2505
EventTableTriggerIO 5864: IOValue=[1], IRC5Controller=? -1, Operator=0, SignalSource=Controlador_IRC5 2505
EventTableTriggerIO 5865: IOValue=[0], IRC5Controller=? -1, Operator=0, SignalSource=Controlador_IRC5 2505
EventTableTriggerIO 5866: IOValue=[1], IRC5Controller=? -1, Operator=0, SignalSource=Controlador_IRC5 2505
EventTableTriggerIO 5867: IOValue=[1], IRC5Controller=? -1, Operator=0, SignalSource=Controlador_IRC5 2505
EventTableTriggerIO 5868: IOValue=[1], IRC5Controller=? -1, Operator=0, SignalSource=Controlador_IRC5 2505
EventTableTriggerIO 5869: IOValue=[1], IRC5Controller=? -1, Operator=0, SignalSource=Controlador_IRC5 2505
EventTableTriggerIO 5870: IOValue=[0], IRC5Controller=? -1, Operator=0, SignalSource=Controlador_IRC5 2505
EventTableTriggerIO 5871: IOValue=[0], IRC5Controller=? -1, Operator=0, SignalSource=Controlador_IRC5 2505
EventTableTriggerIO 5872: IOValue=[0], IRC5Controller=? -1, Operator=0, SignalSource=Controlador_IRC5 2505
EventTableTriggerIO 5873: IOValue=[0], IRC5Controller=? -1, Operator=0, SignalSource=Controlador_IRC5 2505
Targets, tools, work objects and paths stored in the station and not in the controller backup, written as RAPID:
! task T_ROB1
MODULE Module1
  CONST robtarget aprox_verde_arriba_plataf:=[[139.502224541,131.291478687,-27.734922547],[0.27059805,-0.653281482,-0.270598052,-0.653281482],[-1,1,-2,0],[9E+09,9E+09,9E+09,9E+09,9E+09,9E+09]];
ENDMODULE


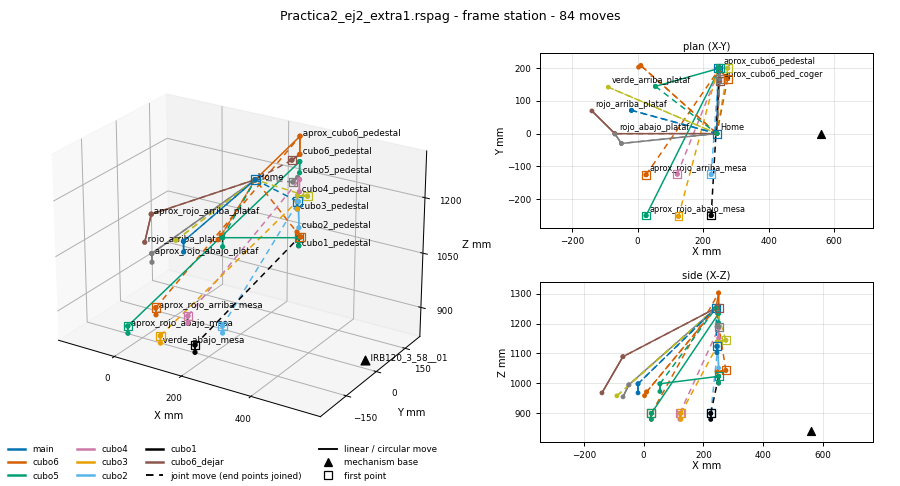
[picture p0: tool path of Practica2_ej2_extra1.rspag in frame station, 84 of 84 moves have a stored position in this frame; points joined in program order, loops and branches not executed]
--- Backups/Controlador_IRC5/RAPID/TASK1/PROGMOD/CalibData.mod ---
MODULE CalibData
	PERS tooldata Pinza_schunk_SGB50_1:=[TRUE,[[-16,0,146.4],[1,0,0,0]],[0.1393,[-13.76,0,75.83],[1,0,0,0],0,0,0]];
    TASK PERS wobjdata WO_Mesa:=[FALSE,TRUE,"",[[107.5,349.842,-0.083],[0.000005,0.999999998,0.000062434,0.000010498]],[[150,25,0],[1,0,0,0]]];
    TASK PERS wobjdata WO_Plataforma:=[FALSE,TRUE,"",[[0,0,0],[1,0,0,0]],[[432.513,-147.487,90],[0,0.92388,0.382683,0]]];
    TASK PERS wobjdata WO_Soporte:=[FALSE,TRUE,"",[[0,0,0],[1,0,0,0]],[[285.003,-175.056,120],[0.00216381,0.999995,0.000457777,0.00216278]]];
ENDMODULE

--- Backups/Controlador_IRC5/RAPID/TASK1/PROGMOD/Module1.mod ---
MODULE Module1
        CONST robtarget aprox_rojo_arriba_mesa:=[[533.94,125.614,59.645],[0,0,1,0],[0,0,0,0],[9E+09,9E+09,9E+09,9E+09,9E+09,9E+09]];
    CONST robtarget rojo_arriba_mesa:=[[533.94,125.614,39.645],[0,0,1,0],[0,0,0,0],[9E+09,9E+09,9E+09,9E+09,9E+09,9E+09]];
    CONST robtarget aprox_cubo6_pedestal:=[[25.549279317,26.09461213,-342.046996466],[0.000457758,0.002162758,0.0021638,-0.999995215],[-1,0,-1,0],[9E+09,9E+09,9E+09,9E+09,9E+09,9E+09]];
    CONST robtarget cubo6_pedestal:=[[25.339411386,25.882309306,-292.826632575],[0.000457758,0.002162758,0.0021638,-0.999995215],[-1,0,-1,0],[9E+09,9E+09,9E+09,9E+09,9E+09,9E+09]];
    CONST robtarget aprox_rojo_abajo_mesa:=[[533.94,250.007672792,59.645],[0,0,1,0],[0,0,0,0],[9E+09,9E+09,9E+09,9E+09,9E+09,9E+09]];
    CONST robtarget rojo_abajo_mesa:=[[533.94,250.007672792,39.645],[0,0,1,0],[0,0,0,0],[9E+09,9E+09,9E+09,9E+09,9E+09,9E+09]];
    CONST robtarget aprox_cubo5_pedestal:=[[25.254654145,25.797431875,-273.222657828],[0.000457758,0.002162758,0.0021638,-0.999995215],[-1,0,-1,0],[9E+09,9E+09,9E+09,9E+09,9E+09,9E+09]];
    CONST robtarget cubo5_pedestal:=[[25.120317008,25.665050592,-242.832912358],[0.000457758,0.002162758,0.0021638,-0.999995215],[-1,0,-1,0],[9E+09,9E+09,9E+09,9E+09,9E+09,9E+09]];
    CONST robtarget aprox_verde_arriba_mesa:=[[438.734213561,123.598213564,60],[0,0.382683432,0.923879533,0],[0,0,0,0],[9E+09,9E+09,9E+09,9E+09,9E+09,9E+09]];
    CONST robtarget verde_arriba_mesa:=[[438.734213561,123.598213564,40],[0,0.382683432,0.923879533,0],[0,0,0,0],[9E+09,9E+09,9E+09,9E+09,9E+09,9E+09]];
    CONST robtarget aprox_cubo4_pedestal:=[[25.040384451,25.585004006,-224.344639308],[0.000457758,0.002162758,0.0021638,-0.999995215],[-1,0,-1,0],[9E+09,9E+09,9E+09,9E+09,9E+09,9E+09]];
    CONST robtarget cubo4_pedestal:=[[24.898685649,25.440965181,-190.890898963],[0.000457758,0.002162758,0.0021638,-0.999995215],[-1,0,-1,0],[9E+09,9E+09,9E+09,9E+09,9E+09,9E+09]];
    CONST robtarget aprox_verde_abajo_mesa:=[[435.029028035,252.504917123,59.645],[0,0.382683431,0.923879533,0],[0,0,0,0],[9E+09,9E+09,9E+09,9E+09,9E+09,9E+09]];
    CONST robtarget verde_abajo_mesa:=[[435.029028035,252.504917123,39.645],[0,0.382683431,0.923879533,0],[0,0,0,0],[9E+09,9E+09,9E+09,9E+09,9E+09,9E+09]];
    CONST robtarget aprox_cubo3_pedestal:=[[30.42096791,25.325653044,-163.237533234],[0.000457758,0.002162758,0.0021638,-0.999995215],[-1,0,-1,0],[9E+09,9E+09,9E+09,9E+09,9E+09,9E+09]];
    CONST robtarget cubo3_pedestal:=[[30.328703887,25.235855903,-142.312757971],[0.000457758,0.002162758,0.0021638,-0.999995215],[-1,0,-1,0],[9E+09,9E+09,9E+09,9E+09,9E+09,9E+09]];
    CONST robtarget aprox_blanco_arriba_mesa:=[[335.341333781,124.646829723,59.645],[0,0,1,0],[0,0,0,0],[9E+09,9E+09,9E+09,9E+09,9E+09,9E+09]];
    CONST robtarget blanco_arriba_mesa:=[[335.341333781,124.646829723,39.645],[0,0,1,0],[0,0,0,0],[9E+09,9E+09,9E+09,9E+09,9E+09,9E+09]];
    CONST robtarget aprox_cubo2_pedestal:=[[27.266373262,25.322794354,-163.251184928],[0.000457758,0.002162758,0.0021638,-0.999995215],[-1,0,-1,0],[9E+09,9E+09,9E+09,9E+09,9E+09,9E+09]];
    CONST robtarget cubo2_pedestal:=[[24.467094805,25.008772287,-91.069146441],[0.000457758,0.002162758,0.0021638,-0.999995215],[-1,0,-1,0],[9E+09,9E+09,9E+09,9E+09,9E+09,9E+09]];
    CONST robtarget aprox_blanco_abajo_mesa:=[[335.341333781,250.007672792,59.645],[0,0,1,0],[0,0,0,0],[9E+09,9E+09,9E+09,9E+09,9E+09,9E+09]];
    CONST robtarget blanco_abajo_mesa:=[[335.341333781,250.007672792,39.645],[0,0,1,0],[0,0,0,0],[9E+09,9E+09,9E+09,9E+09,9E+09,9E+09]];
    CONST robtarget aprox_cubo1_pedestal:=[[24.343935799,24.887581907,-63.263832832],[0.000457758,0.002162758,0.0021638,-0.999995215],[-1,0,-1,0],[9E+09,9E+09,9E+09,9E+09,9E+09,9E+09]];
    CONST robtarget cubo1_pedestal:=[[24.250158502,24.79153128,-40.893706829],[0.000457758,0.002162758,0.0021638,-0.999995215],[-1,0,-1,0],[9E+09,9E+09,9E+09,9E+09,9E+09,9E+09]];
    CONST robtarget aprox_cubo6_ped_coger:=[[25.36309876,-13.151520628,-290.806707862],[0.500227007,-0.49760545,-0.500225966,-0.501932008],[0,1,-1,1],[9E+09,9E+09,9E+09,9E+09,9E+09,9E+09]];
    CONST robtarget cubo6_ped_coger:=[[25.339411386,25.882309306,-292.826632575],[0.500227007,-0.49760545,-0.500225966,-0.501932008],[0,1,-1,1],[9E+09,9E+09,9E+09,9E+09,9E+09,9E+09]];
    CONST robtarget aprox_rojo_arriba_plataf:=[[243.457745108,34.48993352,-159.08793761],[0.499999999,-0.499999999,-0.500000001,-0.500000001],[0,-2,0,0],[9E+09,9E+09,9E+09,9E+09,9E+09,9E+09]];
    CONST robtarget rojo_arriba_plataf:=[[243.906538693,133.195793854,-38.178674671],[0.499999999,-0.500000001,-0.499999999,-0.500000001],[0,-2,0,0],[9E+09,9E+09,9E+09,9E+09,9E+09,9E+09]];
    CONST robtarget Home:=[[318,0,411.6],[0,0,1,0],[0,0,0,0],[9E+09,9E+09,9E+09,9E+09,9E+09,9E+09]];
    CONST robtarget aprox_cubo5_ped_coger:=[[24.911428859,-6.83845608,-229.288823654],[0.500227007,-0.49760545,-0.500225966,-0.501932008],[0,1,-1,1],[9E+09,9E+09,9E+09,9E+09,9E+09,9E+09]];
    CONST robtarget cubo5_ped_coger:=[[30.50939036,25.610734623,-229.124126392],[0.500227007,-0.49760545,-0.500225966,-0.501932008],[0,1,-1,1],[9E+09,9E+09,9E+09,9E+09,9E+09,9E+09]];
    CONST robtarget aprox_rojo_abajo_plataf:=[[250.469249959,-0.607665298,-65.153333948],[0.499999999,-0.499999999,-0.500000001,-0.500000001],[0,-2,1,0],[9E+09,9E+09,9E+09,9E+09,9E+09,9E+09]];
    CONST robtarget rojo_abajo_plataf:=[[244.032373493,33.321628453,-24.989521495],[0.500000001,-0.500000001,-0.499999999,-0.499999999],[0,-2,1,0],[9E+09,9E+09,9E+09,9E+09,9E+09,9E+09]];
    CONST robtarget aprox_cubo4_ped_coger:=[[0.627579609,25.387847835,-183.986772295],[0.001853721,-0.705574097,0.001206354,-0.708632699],[-1,1,-2,0],[9E+09,9E+09,9E+09,9E+09,9E+09,9E+09]];
    CONST robtarget cubo4_ped_coger:=[[30.293212649,25.394256051,-179.125062359],[0.001853721,-0.705574097,0.001206354,-0.708632699],[-1,1,-2,0],[9E+09,9E+09,9E+09,9E+09,9E+09,9E+09]];
    CONST robtarget verde_arriba_plataf:=[[157.376586831,149.165841753,-28.258517858],[0.270598049,-0.653281483,-0.270598049,-0.653281483],[-1,-1,0,1],[9E+09,9E+09,9E+09,9E+09,9E+09,9E+09]];
    CONST robtarget aprox_verde_abajo_plataf:=[[157.376587031,49.165841339,-68.480283741],[0.382683433,0,0,-0.923879532],[-1,0,-1,0],[9E+09,9E+09,9E+09,9E+09,9E+09,9E+09]];
    CONST robtarget verde_abajo_plataf:=[[157.376587031,49.165841753,-38.178674671],[0.382683431,0,0,-0.923879533],[-1,0,-1,0],[9E+09,9E+09,9E+09,9E+09,9E+09,9E+09]];
    CONST robtarget aprox_cubo2_ped_coger:=[[0.221042556,-7.171706916,-83.227310828],[0.500226988,-0.497605444,-0.500225985,-0.501932014],[0,1,-1,1],[9E+09,9E+09,9E+09,9E+09,9E+09,9E+09]];
    CONST robtarget cubo2_ped_coger:=[[29.856964722,24.957400986,-78.226649224],[0.500226988,-0.497605444,-0.500225985,-0.501932014],[0,1,-1,1],[9E+09,9E+09,9E+09,9E+09,9E+09,9E+09]];
    CONST robtarget aprox_blanco_arriba_plataf:=[[40.481081449,125.634648962,-41.100588955],[0.500000001,-0.499999999,-0.500000001,-0.499999999],[-1,-2,1,0],[9E+09,9E+09,9E+09,9E+09,9E+09,9E+09]];
    CONST robtarget blanco_arriba_plataf:=[[48.890339975,126.840686937,-28.68251683],[0.499999999,-0.500000001,-0.499999999,-0.500000001],[-1,-2,1,0],[9E+09,9E+09,9E+09,9E+09,9E+09,9E+09]];
    CONST robtarget aprox_blanco_abajo_plataf:=[[53.876587031,49.165841546,-68.480283741],[-0.000000001,0,0,1],[-1,0,-1,0],[9E+09,9E+09,9E+09,9E+09,9E+09,9E+09]];
    CONST robtarget blanco_abajo_plataf:=[[53.876587031,49.165841546,-42.881436214],[0.000000001,0,0,1],[-1,0,-1,0],[9E+09,9E+09,9E+09,9E+09,9E+09,9E+09]];
!***********************************************************
    !
    ! Módulo:  Module1
    !
    ! Descripción:
    !   <Introduzca la descripción aquí>
    !
    ! Autor: Rubén
    !
    ! Versión: 1.0
    !
    !***********************************************************


    !***********************************************************
    !
    ! Procedimiento Main
    !
    !   Este es el punto de entrada de su programa
    !
    !***********************************************************
    VAR num num_cubos := 3;
    PROC moverCubos()
        IF num_cubos >= 1 THEN
            cubo1;
        ENDIF
        IF num_cubos >= 2 THEN
            cubo2;
        ENDIF
        IF num_cubos >= 3 THEN
            cubo3;
        ENDIF
        IF num_cubos >= 4 THEN
            cubo4;
        ENDIF
        IF num_cubos >= 5 THEN
            cubo5;
        ENDIF
        IF num_cubos >= 6 THEN
            cubo6;
        ENDIF
    ENDPROC

    PROC dejarCubos()
        IF num_cubos >= 6 THEN
            cubo6_dejar;
        ENDIF
        IF num_cubos >= 5 THEN
            cubo5_dejar;
        ENDIF
        IF num_cubos >= 4 THEN
            cubo4_dejar;
        ENDIF
        IF num_cubos >= 3 THEN
            cubo3_dejar;
        ENDIF
        IF num_cubos >= 2 THEN
            cubo2_dejar;
        ENDIF
        IF num_cubos >= 1 THEN
            cubo1_dejar;
        ENDIF
    ENDPROC

    PROC main()
        ! Posición segura
        MoveJ Home, v400, fine, Pinza_schunk_SGB50_1\WObj:=wobj0;

        ! Recoger desde mesa y colocar en pedestal
        moverCubos;

        WaitTime 2;

        ! Recoger desde pedestal y colocar en plataforma
        dejarCubos;

        ! Regresar a Home
        MoveJ Home, v400, fine, Pinza_schunk_SGB50_1\WObj:=wobj0;
    ENDPROC

    PROC cubo6()
        MoveJ aprox_rojo_arriba_mesa,v400,fine,Pinza_schunk_SGB50_1\WObj:=wobj0;
        MoveL rojo_arriba_mesa,v200,fine,Pinza_schunk_SGB50_1\WObj:=wobj0;
        SetDO D16_O,1;
        WaitTime 1;
        MoveL aprox_rojo_arriba_mesa,v400,fine,Pinza_schunk_SGB50_1\WObj:=wobj0;
        MoveJ aprox_cubo6_pedestal,v400,fine,Pinza_schunk_SGB50_1\WObj:=WO_Soporte;
        MoveL cubo6_pedestal,v200,fine,Pinza_schunk_SGB50_1\WObj:=WO_Soporte;
        SetDO D16_O,0;
        WaitTime 1;
        MoveL aprox_cubo6_pedestal,v200,fine,Pinza_schunk_SGB50_1\WObj:=WO_Soporte;
        MoveL Home,v400,fine,Pinza_schunk_SGB50_1\WObj:=wobj0;
    ENDPROC
    PROC cubo5()
        MoveJ aprox_rojo_abajo_mesa,v400,z0,Pinza_schunk_SGB50_1\WObj:=wobj0;
        MoveL rojo_abajo_mesa,v200,fine,Pinza_schunk_SGB50_1\WObj:=wobj0;
        SetDO D16_O,1;
        WaitTime 1;
        MoveL aprox_rojo_abajo_mesa,v400,z0,Pinza_schunk_SGB50_1\WObj:=wobj0;
        MoveL aprox_cubo5_pedestal,v200,fine,Pinza_schunk_SGB50_1\WObj:=WO_Soporte;
        MoveL cubo5_pedestal,v200,fine,Pinza_schunk_SGB50_1\WObj:=WO_Soporte;
        SetDO D16_O,0;
        WaitTime 1;
        MoveL aprox_cubo5_pedestal,v200,fine,Pinza_schunk_SGB50_1\WObj:=WO_Soporte;
    ENDPROC
    PROC cubo4()
        MoveJ aprox_verde_arriba_mesa,v400,fine,Pinza_schunk_SGB50_1\WObj:=wobj0;
        WaitTime 1;
        MoveL verde_arriba_mesa,v1000,z100,Pinza_schunk_SGB50_1\WObj:=wobj0;
        WaitTime 1;
        SetDO D16_O,1;
        WaitTime 1;
        MoveL aprox_verde_arriba_mesa,v400,fine,Pinza_schunk_SGB50_1\WObj:=wobj0;
        MoveJ aprox_cubo4_pedestal,v400,fine,Pinza_schunk_SGB50_1\WObj:=WO_Soporte;
        MoveL cubo4_pedestal,v200,fine,Pinza_schunk_SGB50_1\WObj:=WO_Soporte;
        SetDO D16_O,0;
        WaitTime 1;
        MoveL aprox_cubo4_pedestal,v200,fine,Pinza_schunk_SGB50_1\WObj:=WO_Soporte;
    ENDPROC
    PROC cubo3()
        MoveJ aprox_verde_abajo_mesa,v400,fine,Pinza_schunk_SGB50_1\WObj:=wobj0;
        MoveL verde_abajo_mesa,v200,fine,Pinza_schunk_SGB50_1\WObj:=wobj0;
        SetDO D16_O,1;
        WaitTime 1;
        MoveL aprox_verde_abajo_mesa,v200,fine,Pinza_schunk_SGB50_1\WObj:=wobj0;
        MoveJ aprox_cubo3_pedestal,v400,fine,Pinza_schunk_SGB50_1\WObj:=WO_Soporte;
        MoveL cubo3_pedestal,v200,fine,Pinza_schunk_SGB50_1\WObj:=WO_Soporte;
        SetDO D16_O,0;
        WaitTime 1;
        MoveL aprox_cubo3_pedestal,v400,fine,Pinza_schunk_SGB50_1\WObj:=WO_Soporte;
    ENDPROC
    PROC cubo2()
        MoveJ aprox_blanco_arriba_mesa,v400,fine,Pinza_schunk_SGB50_1\WObj:=wobj0;
        MoveL blanco_arriba_mesa,v200,fine,Pinza_schunk_SGB50_1\WObj:=wobj0;
        SetDO D16_O,1;
        WaitTime 1;
        MoveL aprox_blanco_arriba_mesa,v200,fine,Pinza_schunk_SGB50_1\WObj:=wobj0;
        MoveJ aprox_cubo2_pedestal,v400,fine,Pinza_schunk_SGB50_1\WObj:=WO_Soporte;
        MoveL cubo2_pedestal,v200,fine,Pinza_schunk_SGB50_1\WObj:=WO_Soporte;
        SetDO D16_O,0;
        WaitTime 1;
        MoveL aprox_cubo2_pedestal,v400,fine,Pinza_schunk_SGB50_1\WObj:=WO_Soporte;
    ENDPROC
    PROC cubo1()
        SetDO D16_O,0;
        WaitTime 1;
        MoveJ aprox_blanco_abajo_mesa,v400,fine,Pinza_schunk_SGB50_1\WObj:=wobj0;
        MoveL blanco_abajo_mesa,v200,fine,Pinza_schunk_SGB50_1\WObj:=wobj0;
        SetDO D16_O,1;
        WaitTime 1;
        MoveL aprox_blanco_abajo_mesa,v200,fine,Pinza_schunk_SGB50_1\WObj:=wobj0;
        MoveJ aprox_cubo1_pedestal,v400,fine,Pinza_schunk_SGB50_1\WObj:=WO_Soporte;
        MoveL cubo1_pedestal,v200,fine,Pinza_schunk_SGB50_1\WObj:=WO_Soporte;
        SetDO D16_O,0;
        WaitTime 1;
        MoveL aprox_cubo1_pedestal,v400,fine,Pinza_schunk_SGB50_1\WObj:=WO_Soporte;
    ENDPROC
    PROC cubo6_dejar()
        MoveJ aprox_cubo6_ped_coger,v400,fine,Pinza_schunk_SGB50_1\WObj:=WO_Soporte;
        MoveL cubo6_ped_coger,v200,fine,Pinza_schunk_SGB50_1\WObj:=WO_Soporte;
        SetDO D16_O,1;
        WaitTime 1;
        MoveL aprox_cubo6_ped_coger,v400,fine,Pinza_schunk_SGB50_1\WObj:=WO_Soporte;
        MoveJ Home,v400,fine,Pinza_schunk_SGB50_1\WObj:=wobj0;
        MoveJ aprox_rojo_arriba_plataf,v400,fine,Pinza_schunk_SGB50_1\WObj:=WO_Plataforma;
        MoveL rojo_arriba_plataf,v200,fine,Pinza_schunk_SGB50_1\WObj:=WO_Plataforma;
        SetDO D16_O,0;
        WaitTime 1;
        MoveL aprox_rojo_arriba_plataf,v400,fine,Pinza_schunk_SGB50_1\WObj:=WO_Plataforma;
        MoveL Home,v400,fine,Pinza_schunk_SGB50_1\WObj:=wobj0;
    ENDPROC
    PROC cubo5_dejar()
        MoveJ aprox_cubo5_ped_coger,v400,fine,Pinza_schunk_SGB50_1\WObj:=WO_Soporte;
        MoveL cubo5_ped_coger,v200,fine,Pinza_schunk_SGB50_1\WObj:=WO_Soporte;
        SetDO D16_O,1;
        WaitTime 1;
        MoveL aprox_cubo5_ped_coger,v200,fine,Pinza_schunk_SGB50_1\WObj:=WO_Soporte;
        MoveJ Home,v400,fine,Pinza_schunk_SGB50_1\WObj:=wobj0;
        MoveJ aprox_rojo_abajo_plataf,v400,fine,Pinza_schunk_SGB50_1\WObj:=WO_Plataforma;
        MoveL rojo_abajo_plataf,v200,fine,Pinza_schunk_SGB50_1\WObj:=WO_Plataforma;
        SetDO D16_O,0;
        WaitTime 1;
        MoveL aprox_rojo_abajo_plataf,v200,fine,Pinza_schunk_SGB50_1\WObj:=WO_Plataforma;
        MoveL Home,v400,fine,Pinza_schunk_SGB50_1\WObj:=wobj0;
    ENDPROC
    PROC cubo4_dejar()
        MoveL aprox_cubo4_ped_coger,v200,fine,Pinza_schunk_SGB50_1\WObj:=WO_Soporte;
        MoveL cubo4_ped_coger,v200,fine,Pinza_schunk_SGB50_1\WObj:=WO_Soporte;
        SetDO D16_O,1;
        WaitTime 1;
        MoveL aprox_cubo4_ped_coger,v200,fine,Pinza_schunk_SGB50_1\WObj:=WO_Soporte;
        MoveJ Home,v200,fine,Pinza_schunk_SGB50_1\WObj:=wobj0;
        MoveJ verde_arriba_plataf,v200,fine,Pinza_schunk_SGB50_1\WObj:=WO_Plataforma;
        SetDO D16_O,0;
        WaitTime 1;
        MoveJ Home,v400,fine,Pinza_schunk_SGB50_1\WObj:=wobj0;
    ENDPROC
    PROC cubo3_dejar()
        MoveL aprox_cubo3_pedestal,v400,fine,Pinza_schunk_SGB50_1\WObj:=WO_Soporte;
        MoveL cubo3_pedestal,v400,fine,Pinza_schunk_SGB50_1\WObj:=WO_Soporte;
        SetDO D16_O,1;
        WaitTime 1;
        MoveL aprox_cubo3_pedestal,v400,fine,Pinza_schunk_SGB50_1\WObj:=WO_Soporte;
        MoveJ Home,v200,fine,Pinza_schunk_SGB50_1\WObj:=wobj0;
        MoveJ aprox_verde_abajo_plataf,v400,fine,Pinza_schunk_SGB50_1\WObj:=WO_Plataforma;
        MoveL verde_abajo_plataf,v1000,fine,Pinza_schunk_SGB50_1\WObj:=WO_Plataforma;
        SetDO D16_O,0;
        WaitTime 1;
        MoveL aprox_verde_abajo_plataf,v1000,fine,Pinza_schunk_SGB50_1\WObj:=WO_Plataforma;
        MoveJ Home,v400,fine,Pinza_schunk_SGB50_1\WObj:=wobj0;
    ENDPROC
    PROC cubo2_dejar()
        MoveJ aprox_cubo2_ped_coger,v200,fine,Pinza_schunk_SGB50_1\WObj:=WO_Soporte;
        MoveL cubo2_ped_coger,v200,fine,Pinza_schunk_SGB50_1\WObj:=WO_Soporte;
        SetDO D16_O,1;
        WaitTime 1;
        MoveL aprox_cubo2_ped_coger,v200,fine,Pinza_schunk_SGB50_1\WObj:=WO_Soporte;
        MoveJ Home,v400,fine,Pinza_schunk_SGB50_1\WObj:=wobj0;
        MoveJ aprox_blanco_arriba_plataf,v400,fine,Pinza_schunk_SGB50_1\WObj:=WO_Plataforma;
        MoveL blanco_arriba_plataf,v200,fine,Pinza_schunk_SGB50_1\WObj:=WO_Plataforma;
        SetDO D16_O,0;
        WaitTime 1;
        MoveL aprox_blanco_arriba_plataf,v200,fine,Pinza_schunk_SGB50_1\WObj:=WO_Plataforma;
        MoveJ Home,v400,fine,Pinza_schunk_SGB50_1\WObj:=wobj0;
    ENDPROC
    PROC cubo1_dejar()
        MoveL aprox_cubo1_pedestal,v200,fine,Pinza_schunk_SGB50_1\WObj:=WO_Soporte;
        MoveL cubo1_pedestal,v200,fine,Pinza_schunk_SGB50_1\WObj:=WO_Soporte;
        SetDO D16_O,1;
        WaitTime 1;
        MoveL aprox_cubo1_pedestal,v200,fine,Pinza_schunk_SGB50_1\WObj:=WO_Soporte;
        MoveL aprox_blanco_abajo_plataf,v200,fine,Pinza_schunk_SGB50_1\WObj:=WO_Plataforma;
        MoveL blanco_abajo_plataf,v200,fine,Pinza_schunk_SGB50_1\WObj:=WO_Plataforma;
        SetDO D16_O,0;
        WaitTime 1;
        MoveL aprox_blanco_abajo_plataf,v200,fine,Pinza_schunk_SGB50_1\WObj:=WO_Plataforma;
        MoveJ Home,v400,fine,Pinza_schunk_SGB50_1\WObj:=wobj0;
    ENDPROC
ENDMODULE

--- Backups/Controlador_IRC5/SYSPAR/EIO.cfg ---
EIO:CFG_1.0:6:1::
#
EIO_SIGNAL:

      -Name "D16_O" -SignalType "DO" -Access "All"
